FUNCTION_BLOCK WagoPublishTest (* Composite Function Block Type *)
  (* Standard: 61499-2 *)
  (* Version 0.2, 2003-12-05, JHC, Rockwell Automation, Renamed from NEWCOMPFB. *)
  (* Compiler header: package fb.rt.wago; *)
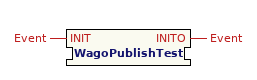
  EVENT_INPUT
    INIT; (* Initialization Request *)
  END_EVENT
  EVENT_OUTPUT
    INITO; (* Initialization Confirm *)
  END_EVENT
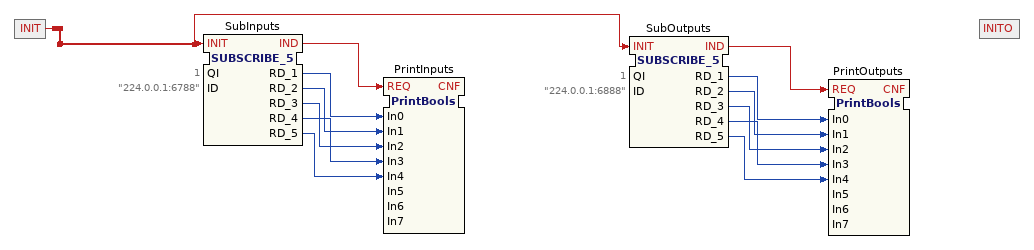
  FBS
    PrintInputs : PrintBools;
    PrintOutputs : PrintBools;
    SubInputs : SUBSCRIBE_5(QI := 1, ID := "224.0.0.1:6788");
    SubOutputs : SUBSCRIBE_5(QI := 1, ID := "224.0.0.1:6888");
  END_FBS
  EVENT_CONNECTIONS
    INIT TO SubInputs.INIT;
    INIT TO SubOutputs.INIT;
    SubInputs.IND TO PrintInputs.REQ;
    SubOutputs.IND TO PrintOutputs.REQ;
  END_CONNECTIONS
  DATA_CONNECTIONS
    SubInputs.RD_1 TO PrintInputs.In0;
    SubInputs.RD_2 TO PrintInputs.In1;
    SubInputs.RD_3 TO PrintInputs.In2;
    SubInputs.RD_4 TO PrintInputs.In3;
    SubInputs.RD_5 TO PrintInputs.In4;
    SubOutputs.RD_1 TO PrintOutputs.In0;
    SubOutputs.RD_2 TO PrintOutputs.In1;
    SubOutputs.RD_3 TO PrintOutputs.In2;
    SubOutputs.RD_4 TO PrintOutputs.In3;
    SubOutputs.RD_5 TO PrintOutputs.In4;
  END_CONNECTIONS
END_FUNCTION_BLOCK
